PROGRAM Axis_01_Function_Blocks
VAR
END_VAR

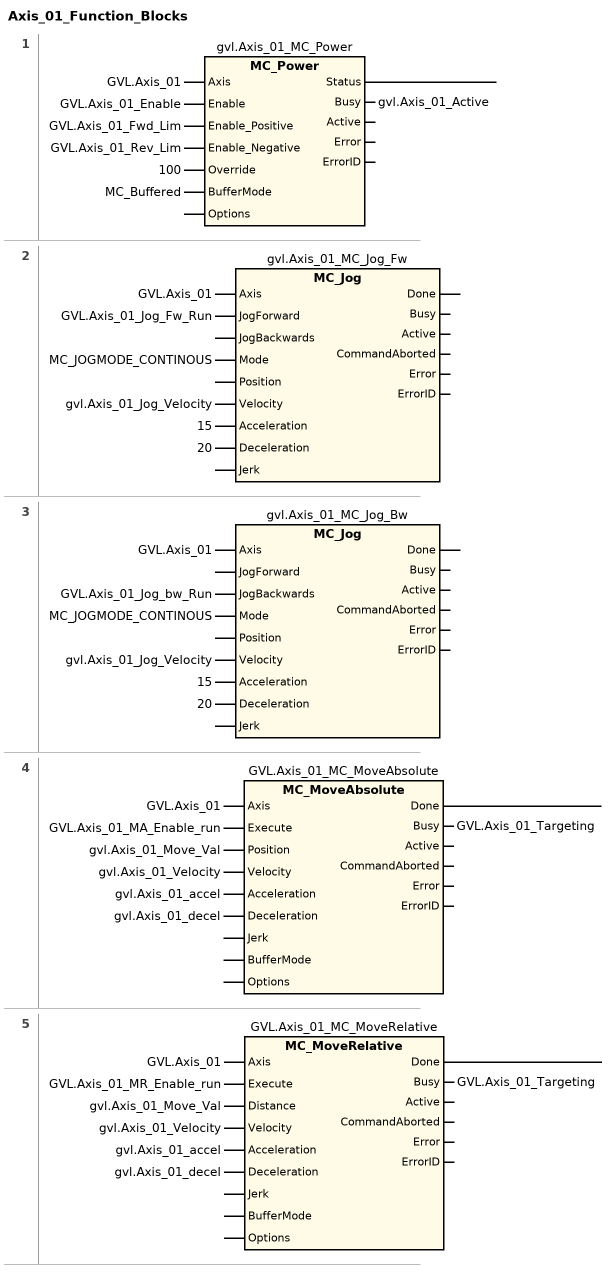
// NETWORK 1
gvl.Axis_01_MC_Power(
    Axis := GVL.Axis_01,
    Enable := GVL.Axis_01_Enable,
    Enable_Positive := GVL.Axis_01_Fwd_Lim,
    Enable_Negative := GVL.Axis_01_Rev_Lim,
    Override := 100,
    BufferMode := MC_Buffered,
    Busy => gvl.Axis_01_Active); // MC_Power

// NETWORK 2
gvl.Axis_01_MC_Jog_Fw(
    Axis := GVL.Axis_01,
    JogForward := GVL.Axis_01_Jog_Fw_Run,
    Mode := MC_JOGMODE_CONTINOUS,
    Velocity := gvl.Axis_01_Jog_Velocity,
    Acceleration := 15,
    Deceleration := 20); // MC_Jog

// NETWORK 3
gvl.Axis_01_MC_Jog_Bw(
    Axis := GVL.Axis_01,
    JogBackwards := GVL.Axis_01_Jog_bw_Run,
    Mode := MC_JOGMODE_CONTINOUS,
    Velocity := gvl.Axis_01_Jog_Velocity,
    Acceleration := 15,
    Deceleration := 20); // MC_Jog

// NETWORK 4
GVL.Axis_01_MC_MoveAbsolute(
    Axis := GVL.Axis_01,
    Execute := GVL.Axis_01_MA_Enable_run,
    Position := gvl.Axis_01_Move_Val,
    Velocity := gvl.Axis_01_Velocity,
    Acceleration := gvl.Axis_01_accel,
    Deceleration := gvl.Axis_01_decel,
    Busy => GVL.Axis_01_Targeting); // MC_MoveAbsolute

// NETWORK 5
GVL.Axis_01_MC_MoveRelative(
    Axis := GVL.Axis_01,
    Execute := GVL.Axis_01_MR_Enable_run,
    Distance := gvl.Axis_01_Move_Val,
    Velocity := gvl.Axis_01_Velocity,
    Acceleration := gvl.Axis_01_accel,
    Deceleration := gvl.Axis_01_decel,
    Busy => GVL.Axis_01_Targeting); // MC_MoveRelative

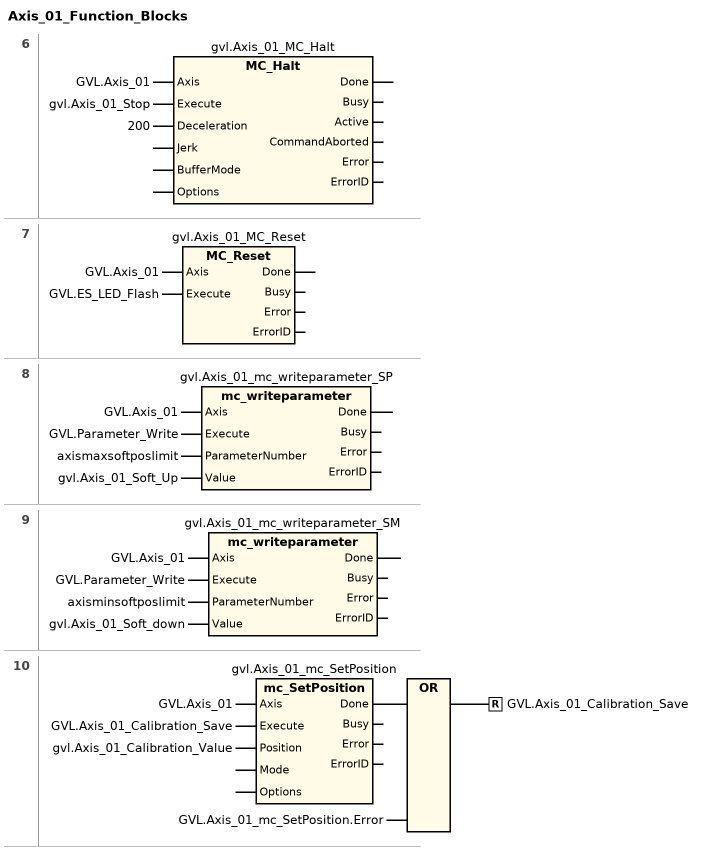
// NETWORK 6
gvl.Axis_01_MC_Halt(Axis := GVL.Axis_01, Execute := gvl.Axis_01_Stop, Deceleration := 200); // MC_Halt

// NETWORK 7
gvl.Axis_01_MC_Reset(Axis := GVL.Axis_01, Execute := GVL.ES_LED_Flash); // MC_Reset

// NETWORK 8
gvl.Axis_01_mc_writeparameter_SP(
    Axis := GVL.Axis_01,
    Execute := GVL.Parameter_Write,
    ParameterNumber := axismaxsoftposlimit,
    Value := gvl.Axis_01_Soft_Up); // mc_writeparameter

// NETWORK 9
gvl.Axis_01_mc_writeparameter_SM(
    Axis := GVL.Axis_01,
    Execute := GVL.Parameter_Write,
    ParameterNumber := axisminsoftposlimit,
    Value := gvl.Axis_01_Soft_down); // mc_writeparameter

// NETWORK 10
gvl.Axis_01_mc_SetPosition(
    Axis := GVL.Axis_01,
    Execute := GVL.Axis_01_Calibration_Save,
    Position := gvl.Axis_01_Calibration_Value); // mc_SetPosition
GVL.Axis_01_Calibration_Save R= gvl.Axis_01_mc_SetPosition.Done OR GVL.Axis_01_mc_SetPosition.Error;

END_PROGRAM

(* stored: Version 1.1.0.1, ProductVersion 3.1.4024.3
   POU Axis_01_Function_Blocks: Id {f2477c3e-db55-4e97-a6e4-f4f2a68821da}, SpecialFunc None *)
